// TIA Portal V17 export
// export: Created 2022-07-20T06:59:47.4747821Z, ExportSetting WithDefaults, DisplayName Totally Integrated Automation Portal, DisplayVersion V17, DisplayName TIA Portal Openness, DisplayVersion V17, DisplayName TIA Portal Version Control Interface, DisplayVersion V17, DisplayName SINAMICS Startdrive Advanced, DisplayVersion V17, DisplayName SINAMICS Startdrive G130, G150, S120, S150, SINAMICS MV, S210, DisplayVersion V17, DisplayName SINAMICS Startdrive G110M, G120, G120C, G120D, G120P, G115D, DisplayVersion V17, DisplayName STEP 7 Professional, DisplayVersion V17, DisplayName STEP 7 Safety, DisplayVersion V17, DisplayName WinCC Advanced, DisplayVersion V17
FUNCTION_BLOCK "FB10120_SinamicsV20_Modbus"   // FB10120, LAD
TITLE = FB10120_SinamicsV20_Modbus
{ S7_Optimized_Access := 'TRUE' }
AUTHOR : Anirouddh
FAMILY : 1012x_SINAMICS_V20
VERSION : 1.0
// Release note : 
// 1.0 - Feature developped
// stored: AutoNumber false, IsIECCheckEnabled false, IsRetainMemResEnabled false, MemoryReserve 100, SetENOAutomatically false, UDAEnableTagReadback false
   VAR_INPUT
      MotorInError : Bool;
      SpeedSetpoint : Real := 200.0;   // mm/s
      AxisDiameter { ExternalAccessible := 'False'; ExternalVisible := 'False'; ExternalWritable := 'False'} : Real := 84.0;   // (mm)
      Gear : Real := 12.5;   // Ratio
      RequestAcknowledge : Bool;
      MotorMaxSpeedRotation { ExternalAccessible := 'False'; ExternalVisible := 'False'; ExternalWritable := 'False'} : Int := 1600;   // (tr/min)
      RequestChangeSpeed : Bool;
      RequestStartMotor : Bool;
      ModbusRtuRequestDone : Bool;
   END_VAR
   VAR_OUTPUT
      StartMotor : Bool;
      AlarmReset : Bool;
      MotorStarted : Bool;
      MotorStopped : Bool;
      StartModbusRtuCommunication : Bool;
      ModbusRtuDataAddress : UInt;
      ModbusRtuDataLength : UInt;
      ModbusRtuMode : USInt;
      ModbusRtuDataRegisterToSend : Int;
      ModbusRtuDataRegisterToSend_1 : Int;
      ReadAlarmCodeDone : Bool;
      SpeedChangeDone : Bool;
      MaterialOk : Bool;
   END_VAR
   VAR
      RequestMotorStartUp : Bool;
      MaximalSpeed : Real;   // mm/s
      SpeedSetPoint_1 : Real;
      ModbusCommunicationStateDiagram : Int;
      MotorStartUpStateDiagram : Int;
      MotorMovementStateDiagram : Int;
      MotorAlarmManagementStateDiagram : Int;
      SpeedSetPointMemory : Real;
      R_TRIG_Start : R_TRIG;
      R_TRIG_RequestChangeSpeed { S7_SetPoint := 'True'} : R_TRIG;
      R_TRIG_RequestAcknowledge { S7_SetPoint := 'True'} : R_TRIG;
      F_TRIG_Start : F_TRIG;
      F_TRIG_MotorInError { S7_SetPoint := 'True'} : F_TRIG;
      TON_StartMotorSignal { S7_SetPoint := 'True'} : TON_TIME;
      TON_StopMotorSignal { S7_SetPoint := 'True'} : TON_TIME;
      TON_AlarmResetSignal { S7_SetPoint := 'True'} : TON_TIME;
   END_VAR
   VAR CONSTANT
      Pi : Real := 3.141592;
      WAIT_FOR_MOTOR_START_UP : Int := 0;
      INITIALIZE_SPEED : Int := 10;
      MOTOR_START_UP_DONE : Int := 20;
      "==========" : Bool;
      WAIT_FOR_MODBUS_COMMUNICATION_REQUEST : Int := 0;
      WRITE_SPEED_SET_POINT : Int := 10;
      MODBUS_COMMUNICATION_DONE : Int := 20;
      "==========_1" : Bool;
      WAIT_FOR_MOVEMENT_REQUEST : Int := 0;
      START_BELT : Int := 20;
      STOP_BELT : Int := 30;
      MOVEMENT_DONE : Int := 50;
      "==========_2" : Bool;
      WAIT_FOR_MOTOR_ERROR : Int := 0;
      RESET_MOTOR_COMMUNICATION_MOVEMENT : Int := 10;
      ALARM_RESET : Int := 20;
      GATHER_ERROR_CODE : Int := 30;
      MOTOR_ERROR_MANAGEMENT_DONE : Int := 40;
   END_VAR
BEGIN

REGION Network 1 (SCL): First Scan
   IF "FirstScan" THEN
       #RequestMotorStartUp := TRUE;
       #SpeedSetPointMemory := 0.0;
       #ModbusCommunicationStateDiagram := 0;
       #SpeedChangeDone := FALSE;
       #ReadAlarmCodeDone := FALSE;
   END_IF;
END_REGION

REGION Network 2 (SCL): Maximum Speed Calculation
   #MaximalSpeed := ((#Pi*#AxisDiameter / #Gear) * (#MotorMaxSpeedRotation))/60;
END_REGION

REGION Network 3 (SCL): %Speed Setpoint Calculation
   #SpeedSetPoint_1 := (#SpeedSetpoint * (100 / #MaximalSpeed));
END_REGION

REGION Network 4 (SCL): Motor Start Up Management
   CASE #MotorStartUpStateDiagram OF
       #WAIT_FOR_MOTOR_START_UP:
           IF #RequestMotorStartUp AND #RequestAcknowledge THEN
               #MotorStartUpStateDiagram := #INITIALIZE_SPEED;
           END_IF;
       #INITIALIZE_SPEED:
           #ModbusRtuDataRegisterToSend.%X0 := #RequestStartMotor;  //Start
           #ModbusRtuDataRegisterToSend.%X1 := TRUE;   //Electric Stop 
           #ModbusRtuDataRegisterToSend.%X2 := TRUE;   //Quick Stop
           #ModbusRtuDataRegisterToSend.%X3 := TRUE;   //Allow Pulse
           #ModbusRtuDataRegisterToSend.%X4 := TRUE;   //Allow GR
           #ModbusRtuDataRegisterToSend.%X5 := TRUE;   //Start GR
           #ModbusRtuDataRegisterToSend.%X6 := TRUE;   //Start Setpoint
           #ModbusRtuDataRegisterToSend.%X7 := FALSE;  //Allow Acknowledge
           #ModbusRtuDataRegisterToSend.%X8 := FALSE;  //JOG Right
           #ModbusRtuDataRegisterToSend.%X9 := FALSE;  //JOG left 
           #ModbusRtuDataRegisterToSend.%X10 := TRUE;  //PLC Control
           #ModbusRtuDataRegisterToSend_1 := REAL_TO_INT(#SpeedSetPoint_1 * 163.84 * 1.12); // SpeedSetPoint * ? * Correction
           #StartModbusRtuCommunication := TRUE;
           #ModbusRtuDataAddress := 40100;
           #ModbusRtuDataLength := 2;
           #ModbusRtuMode := "MODBUS_RTU_WRITE_MODE";
           IF #ModbusRtuRequestDone THEN
               #StartModbusRtuCommunication := FALSE;
               #MotorStartUpStateDiagram := #MOTOR_START_UP_DONE;
           END_IF;
       #MOTOR_START_UP_DONE:
           #MaterialOk := TRUE;
           #RequestMotorStartUp := FALSE;
   END_CASE;
END_REGION

REGION Network 5 (SCL): Motor Communication Managemnt
   CASE #ModbusCommunicationStateDiagram OF
       #WAIT_FOR_MODBUS_COMMUNICATION_REQUEST:
           #R_TRIG_RequestChangeSpeed(CLK := #RequestChangeSpeed);
           IF #R_TRIG_RequestChangeSpeed.Q THEN
               #SpeedChangeDone := FALSE;
               #ModbusCommunicationStateDiagram := #WRITE_SPEED_SET_POINT;
           END_IF;
       #WRITE_SPEED_SET_POINT:
           #ModbusRtuDataRegisterToSend.%X0 := #RequestStartMotor;  //Start
           #ModbusRtuDataRegisterToSend.%X1 := TRUE;   //Electric Stop 
           #ModbusRtuDataRegisterToSend.%X2 := TRUE;   //Quick Stop
           #ModbusRtuDataRegisterToSend.%X3 := TRUE;   //Allow Pulse
           #ModbusRtuDataRegisterToSend.%X4 := TRUE;   //Allow GR
           #ModbusRtuDataRegisterToSend.%X5 := TRUE;   //Start GR
           #ModbusRtuDataRegisterToSend.%X6 := TRUE;   //Start Setpoint
           #ModbusRtuDataRegisterToSend.%X7 := FALSE;  //Allow Acknowledge
           #ModbusRtuDataRegisterToSend.%X8 := FALSE;  //JOG Right
           #ModbusRtuDataRegisterToSend.%X9 := FALSE;  //JOG left 
           #ModbusRtuDataRegisterToSend.%X10 := TRUE;  //PLC Control
           #ModbusRtuDataRegisterToSend_1 := REAL_TO_INT(#SpeedSetPoint_1 * 163.84 * 1.12); // SpeedSetPoint * ? * Correction
           #StartModbusRtuCommunication := TRUE;
           #ModbusRtuDataAddress := 40100;
           #ModbusRtuDataLength := 2;
           #ModbusRtuMode := "MODBUS_RTU_WRITE_MODE";
           IF #ModbusRtuRequestDone THEN
               #SpeedChangeDone := TRUE;
               #StartModbusRtuCommunication := FALSE;
               #ModbusCommunicationStateDiagram := #MODBUS_COMMUNICATION_DONE;
           END_IF;
       #MODBUS_COMMUNICATION_DONE:
           #ModbusCommunicationStateDiagram := #WAIT_FOR_MODBUS_COMMUNICATION_REQUEST;
   END_CASE;
END_REGION

REGION Network 6 (SCL): Motor Movement Management
   CASE #MotorMovementStateDiagram OF
       #WAIT_FOR_MOVEMENT_REQUEST:
           #R_TRIG_Start(CLK := #RequestStartMotor);
           #F_TRIG_Start(CLK := #RequestStartMotor);
           IF #R_TRIG_Start.Q THEN
               #MotorStarted := FALSE;
               #MotorStopped := FALSE;
               #ReadAlarmCodeDone := FALSE;
               #MotorMovementStateDiagram := #START_BELT;
           ELSIF #F_TRIG_Start.Q THEN
               #MotorStarted := FALSE;
               #MotorStopped := FALSE;
               #ReadAlarmCodeDone := FALSE;
               #MotorMovementStateDiagram := #STOP_BELT;
           END_IF;
       #START_BELT:
               #StartMotor := TRUE;
               IF #TON_StartMotorSignal.Q THEN
                   RESET_TIMER(#TON_StartMotorSignal);
                   #MotorStarted := TRUE;
                   #MotorMovementStateDiagram := #MOVEMENT_DONE;
               END_IF;
           #STOP_BELT:
               #StartMotor := FALSE;
               IF #TON_StopMotorSignal.Q THEN
                   #MotorStopped := FALSE;
                   RESET_TIMER(#TON_StopMotorSignal);
                   #MotorMovementStateDiagram := #MOVEMENT_DONE;
               END_IF;
       #MOVEMENT_DONE:
           #MotorMovementStateDiagram := #WAIT_FOR_MOVEMENT_REQUEST;
   END_CASE;
END_REGION

REGION Network 7 (SCL): Motor Error Management
   CASE #MotorAlarmManagementStateDiagram OF
       #WAIT_FOR_MOTOR_ERROR:
           #F_TRIG_MotorInError(CLK := #MotorInError);
           #R_TRIG_RequestAcknowledge(CLK := #RequestAcknowledge);
           IF #F_TRIG_MotorInError.Q THEN
               #ReadAlarmCodeDone := FALSE;
               #MotorAlarmManagementStateDiagram := #RESET_MOTOR_COMMUNICATION_MOVEMENT;
           ELSIF #R_TRIG_RequestAcknowledge.Q THEN
               #ReadAlarmCodeDone := FALSE;
               #MotorAlarmManagementStateDiagram := #ALARM_RESET;
           END_IF;
       #RESET_MOTOR_COMMUNICATION_MOVEMENT:
           #ModbusCommunicationStateDiagram := #WAIT_FOR_MODBUS_COMMUNICATION_REQUEST;
           #MotorMovementStateDiagram := #WAIT_FOR_MOVEMENT_REQUEST;
           #StartMotor := FALSE;
           IF (#ModbusCommunicationStateDiagram = #WAIT_FOR_MODBUS_COMMUNICATION_REQUEST) AND (#MotorMovementStateDiagram = #WAIT_FOR_MOVEMENT_REQUEST) AND NOT (#StartModbusRtuCommunication) THEN
               #MotorAlarmManagementStateDiagram := #GATHER_ERROR_CODE;
           END_IF;
       #ALARM_RESET:
           #AlarmReset := TRUE;
           IF #TON_AlarmResetSignal.Q THEN
               #AlarmReset := FALSE;
               #MotorAlarmManagementStateDiagram := #GATHER_ERROR_CODE;
           END_IF;
       #GATHER_ERROR_CODE:
           #MotorAlarmManagementStateDiagram := #MOTOR_ERROR_MANAGEMENT_DONE;
       #MOTOR_ERROR_MANAGEMENT_DONE:
           #MotorAlarmManagementStateDiagram := #WAIT_FOR_MOTOR_ERROR;
   END_CASE;
END_REGION

REGION Network 8 (SCL): Signal Timers
   //StartSignal
   #TON_StartMotorSignal(IN := #MotorMovementStateDiagram = #START_BELT,
                         PT := T#500ms);

   //StopSignal
   #TON_StopMotorSignal(IN := #MotorMovementStateDiagram = #STOP_BELT,
                        PT := T#500ms);

   //AlarmResetSignal
   #TON_AlarmResetSignal(IN := #MotorAlarmManagementStateDiagram = #ALARM_RESET,
                         PT := T#500ms);
END_REGION
END_FUNCTION_BLOCK
